R_TRIG_1(CLK := hmi_Manual_cal); // R_TRIG
Corrected_count := _w1;
Zero_count := _w2;
Zero_depth_count := Roll_over_count / 2;
IF _w3 THEN (* Corrected_count + Roll_over_count; result not used *) END_IF
IF Corrected_count > (Roll_over_count - Zero_depth_count) THEN (* Corrected_count - Roll_over_count; result not used *) END_IF
R_TRIG_0(CLK := Manual_cal); // R_TRIG
IF R_TRIG_0.Q OR R_TRIG_1.Q THEN _w2 := Count; END_IF
_w1 := Count - Zero_count;
_w3 := Corrected_count < (-Zero_depth_count);
END_METHOD

METHOD M_Depth_history
VAR_INPUT
END_VAR
VAR_INST // added by the converter: edge detectors and wires of the graphical bodies
    _w1, _w2, _w6, _w7 : REAL;
    _w3, _w4 : ANY;
    _w5, _w8 : BOOL;
END_VAR
IF New_depth THEN _w1 := Raw_depth; END_IF
Scan_count := _w2;
IF Late_depth THEN _w3 := 1; END_IF
IF New_depth THEN _w4 := ROL(Depth_history, 1); END_IF
Late_depth := _w5;
_w6 := Raw_depth;
Scan_count := _w7;
New_depth := _w8;
Raw_depth_prev := _w3;
IF NOT New_depth THEN _w2 := Raw_depth + Raw_depth_prev; END_IF
IF New_depth THEN _w7 := 0; END_IF
Depth_history[0] := _w1;
_w5 := Scan_count = Scans_per_update;
_w8 := Raw_depth <> Raw_depth_prev;
Raw_depth_prev := _w6;
Depth_history := _w4;
END_METHOD

METHOD M_Direction
VAR_INPUT
END_VAR
VAR_INST // added by the converter: edge detectors and wires of the graphical bodies
    _w1, _w2, _w3 : REAL;
    _w4, _w5, _w6, _w7, _w9 : BOOL;
    _w8, _w10 : ANY;
END_VAR
Max_pos_reached := _w1;
Max_pos_reached := _w2;
_w3 := Max_pos_reached + Direction_hysteresis;
_w4 := Raw_depth > Max_pos_reached;
IF Going_up AND _w5 THEN _w1 := Raw_depth; END_IF
_w5 := Raw_depth < Max_pos_reached;
_w7 := Going_up AND _w6;
_w6 := Raw_depth > _w3;
IF NOT Going_up AND _w4 THEN _w2 := Raw_depth; END_IF
SR_0(SET1 := _w8, RESET := _w7); // SR
_w8 := NOT Going_up AND _w9;
_w9 := Raw_depth < _w10;
Going_up := SR_0.Q1;
_w10 := Max_pos_reached - Direction_hysteresis;
END_METHOD

METHOD M_Encoder_cal
VAR_INPUT
END_VAR
VAR_INST // added by the converter: edge detectors and wires of the graphical bodies
    _w1, _w3, _w6 : REAL;
    _w2, _w9, _w10, _w11 : ANY;
    _w4, _w5, _w7, _w8 : BOOL;
END_VAR
_w1 := Cal_switch_depth + Cal_window_down;
Offset := _w3;
_w5 := _w4 AND Calibrate AND NOT Rope_capping_mode;
Open_below := Raw_depth > _w2 AND NOT Calibrate AND NOT Rope_capping_mode;
F_TRIG_0(CLK := Calibrate); // F_TRIG
IF F_TRIG_0.Q THEN _w6 := Raw_depth; END_IF
Closed_above := _w5;
Captured_depth := _w6;
_w8 := Captured_depth >= Cal_switch_depth - Cal_window_up AND F_TRIG_0.Q AND _w7 AND NOT Disallow_multiple_cal;
_w7 := Captured_depth <= _w1;
IF _w8 THEN _w3 := _w9; END_IF
_w9 := Cal_switch_depth - Captured_depth;
_w2 := Cal_switch_depth + Cal_window_down;
RS_0(SET := F_TRIG_0.Q, RESET1 := _w10); // RS
_w10 := Raw_depth > _w1;
_w4 := Raw_depth < _w11;
_w11 := Cal_switch_depth - Cal_window_up;
Disallow_multiple_cal := RS_0.Q1;
END_METHOD

METHOD M_Encoder_depth
VAR_INPUT
END_VAR
VAR_INST // added by the converter: edge detectors and wires of the graphical bodies
    _w1, _w2, _w4 : BOOL;
    _w3, _w6, _w7 : REAL;
    _w5 : ANY;
END_VAR
_w2 := ((-Offset) > Cal_window_up OR _w1) + NOT Rope_capping_mode;
_w3 := Raw_depth + Offset;
_w4 := Raw_depth > Max_depth;
Raw_depth := _w6;
Raw_depth := _w5 + NOT Rope_capping_mode;
Encoder_mm := _w7;
_w6 := Encoder_mm + Manual_cal_depth;
_w1 := Offset > Cal_window_down;
_w5 := Min_depth > Raw_depth OR _w4;
Offset_out_of_range := _w2;
Raw_depth := LIMIT(Min_depth, Raw_depth, Max_depth);
_w7 := Corrected_count * mm_per_count;
Calibrated_depth := _w3;
END_METHOD

METHOD M_HMI_command
VAR_INPUT
END_VAR
FB_WORD_TO_BIT_V0_0(Word_in := hmi_Data.Status); // FB_WORD_TO_BIT_V0
hmi_Manual_cal := FB_WORD_TO_BIT_V0_0.bit0;
END_METHOD

METHOD M_HMI_data
VAR_INPUT
END_VAR
VAR_INST // added by the converter: edge detectors and wires of the graphical bodies
    _w1, _w2 : REAL;
    _w3 : ANY;
END_VAR
hmi_data.Status := FB_BIT_TO_WORD_V0_0.Word_out;
_w1 := Count;
_w2 := Raw_depth;
FB_BIT_TO_WORD_V0_0(bit1 := Going_up, bit2 := Movement_detect, bit3 := Calibrate); // FB_BIT_TO_WORD_V0
hmi_data.Calibrated_depth := _w3;
hmi_data.Status := _w1;
hmi_data.Compensated_depth := Compensated_depth;
hmi_data.Raw_depth := _w2;
_w3 := Calibrated_depth;
hmi_data.Raw_count := Raw_count;
hmi_data.Speed := Speed;
END_METHOD

METHOD M_Layering_compensation
VAR_INPUT
END_VAR
VAR_INST // added by the converter: edge detectors and wires of the graphical bodies
    _w1 : REAL;
    _w2 : ANY;
END_VAR
Compensation := _w1;
_w1 := _w2 * Mid_wind_error;
// Add the compensation to the calibrated depth.
Compensated_depth := Calibrated_depth + Compensation;
// Calculate approximate error caused by rope layering. The error should be calibrated to zero at Wind_top_depth and Wind_bottom depth.
// The maximum error should occur roughly at mid-wind (Mid_wind_error). The error is approximated using a sine function.
_w2 := SIN(((Calibrated_depth - Wind_top_depth) / (Wind_bottom_depth - Wind_top_depth)) * 3.14159265);
END_METHOD

METHOD M_Movement_detect
VAR_INPUT
END_VAR
VAR_INST // added by the converter: edge detectors and wires of the graphical bodies
    _w1 : ANY;
    _w2 : REAL;
END_VAR
Movement_detect := RS_1.Q1;
TON_0(IN := Brakes_proved_on, PT := t#500ms); // TON
Brakes_proved_on_500ms := TON_0.Q;
RS_1(SET := ABS(Raw_depth - Brakes_on_depth) > Movement_detect_dist, RESET1 := _w1); // RS
R_TRIG_2(CLK := Brakes_proved_on_500ms); // R_TRIG
_w1 := R_TRIG_2.Q OR Winder_reset;
IF _w1 THEN _w2 := Raw_depth; END_IF
Brakes_on_depth := _w2;
END_METHOD

METHOD M_Speed
VAR_INPUT
END_VAR
VAR
	fbGetCurTaskIdx  : GETCURTASKINDEX;
END_VAR
{warning 'TODO: Task info cycle time is being converted from UDINT to REAL with possible data loss.'}
Speed := (Depth_history[0] - Depth_history[Speed_ave_intervals]) * 1000 
	/ (_TaskInfo[fbGetCurTaskIdx.index].CycleTime * Scans_per_update * Speed_ave_intervals);
END_METHOD

END_FUNCTION_BLOCK

// ---- POUs/FBs/FB_Fast_brake.TcPOU
FUNCTION_BLOCK FB_Fast_brake
VAR_INPUT
	Lh_depth:REAL;
	Rh_depth:REAL;
	Speed:REAL;
	Fast_brake_top_depth:REAL;
	Fast_brake_bottom_depth:REAL;
	Fast_brake_speed:REAL;
	Speed_hysteresis:REAL;
	Off_delay_after_brakes_on:TIME;
	Check_speed:REAL;
END_VAR
VAR_OUTPUT
	Valve:BOOL;
	Active_above_check_speed:BOOL;
END_VAR
VAR
	FB_CTRL_HYSTERESIS_0: FB_CTRL_HYSTERESIS;
	TON_0: TON;
END_VAR

M_Fast_brake();

METHOD M_Fast_brake
VAR_INPUT
END_VAR
{warning 'TODO: HYSTERESIS block needs to be figured out and made to work correctly.'}
VAR_INST // added by the converter: edge detectors and wires of the graphical bodies
    _w1, _w2, _w3, _w4, _w5, _w7 : BOOL;
    _w6 : ANY;
END_VAR
_w1 := Rh_depth <= Fast_brake_top_depth;
_w2 := Lh_depth >= Fast_brake_bottom_depth;
// Lockout if fast brake valve is enabled above check speed
_w3 := Rh_depth >= Fast_brake_bottom_depth;
Active_above_check_speed := (ABS(Speed)) >= Check_speed AND Valve;
_w6 := _w4 AND NOT TON_0.Q AND NOT _w5;
_w5 := (ABS(Speed)) >= 300;
TON_0(IN := Brakes.Proved_on, PT := Off_delay_after_brakes_on); // TON
// Fast braking
FB_CTRL_HYSTERESIS_0(); // FB_CTRL_HYSTERESIS
_w4 := NOT FB_CTRL_HYSTERESIS_0.bOut AND Safety.Sc1 AND Safety.Sc2 OR NOT Clutch.Lh_in OR NOT Clutch.Rh_in OR _w7 OR _w1 OR _w2 OR _w3;
Valve := _w6;
_w7 := Lh_depth <= Fast_brake_top_depth;
END_METHOD

END_FUNCTION_BLOCK

// ---- POUs/FBs/FB_Least_gate_element.TcPOU
FUNCTION_BLOCK FB_Least_gate_element
VAR_INPUT
	Enforce:BOOL;
	Enforce_in_rope_cap:BOOL;
	Allowed_speed:REAL;
	Description:STRING[32];
END_VAR
VAR_OUTPUT
END_VAR
VAR_IN_OUT
	Least_gate_data:dut_Least_gate;
END_VAR
VAR
END_VAR

M_Least_gate_element();

METHOD M_Least_gate_element
VAR_INPUT
END_VAR
VAR_INST // added by the converter: edge detectors and wires of the graphical bodies
    _w1, _w4, _w5 : BOOL;
    _w2, _w3 : ANY;
    _w6 : REAL;
END_VAR
IF _w1 THEN _w2 := Description; END_IF
_w4 := Allowed_speed < _w3;
_w3 := BOOL_TO_REAL(Least_gate_data.Rope_cap_mode);
_w1 := _w4 AND Enforce AND NOT _w5;
IF _w1 THEN _w6 := Allowed_speed; END_IF
Least_gate_data.Min_allowed_speed := _w6;
_w5 := Least_gate_data.Rope_cap_mode AND NOT Enforce_in_rope_cap;
Least_gate_data.Description := _w2;
END_METHOD

END_FUNCTION_BLOCK

// ---- POUs/FBs/FB_Least_gate_result.TcPOU
FUNCTION_BLOCK FB_Least_gate_result
VAR_INPUT
	Rope_cap_mode:BOOL;
END_VAR
VAR_OUTPUT
	Allowed_speed:REAL;
	Description:STRING[32];
END_VAR
VAR_IN_OUT
	Least_gate_data:dut_Least_gate;
END_VAR
VAR
END_VAR

M_Least_gate_result();

METHOD M_Least_gate_result
VAR_INPUT
END_VAR
VAR_INST // added by the converter: edge detectors and wires of the graphical bodies
    _w1, _w2 : ANY;
END_VAR
Least_gate_data.Min_allowed_speed := _w1;
Description := _w2;
_w2 := Least_gate_data.Description;
_w1 := 32000;
Allowed_speed := Least_gate_data.Min_allowed_speed;
Least_gate_data.Description := '';
Least_gate_data.Rope_cap_mode := Rope_cap_mode;
END_METHOD

END_FUNCTION_BLOCK

// ---- POUs/FBs/FB_Mode.TcPOU
FUNCTION_BLOCK FB_Mode
VAR_INPUT
	Men:BOOL;
	Material:BOOL;
	Rock:BOOL;
	Manual_switch:BOOL;
	Auto_switch:BOOL;
	Rope_capping_switch:BOOL;
	Brake_maint_switch:BOOL;
	Single_lever_control:BOOL;
END_VAR
VAR_OUTPUT
	cs_Mode_change:BOOL;
	cs_Men_rock_sw_fault:BOOL;
	cs_Auto_manual_sw_fault:BOOL;
	cs_Men_to_rock:BOOL;
	cs_Rock_to_men:BOOL;
	cs_Auto_to_manual:BOOL;
	cs_Manual_to_auto:BOOL;
	cs_Rope_capping_on:BOOL;
	cs_Rope_capping_off:BOOL;
	cs_Brake_maint_on:BOOL;
	cs_Brake_maint_off:BOOL;
	hmi_Status:WORD;
END_VAR
VAR
	F_TRIG_0: F_TRIG;
	R_TRIG_0: R_TRIG;
	R_TRIG_1: R_TRIG;
	F_TRIG_1: F_TRIG;
	R_TRIG_2: R_TRIG;
	F_TRIG_2: F_TRIG;
	R_TRIG_3: R_TRIG;
	F_TRIG_3: F_TRIG;
	R_TRIG_4: R_TRIG;
	F_TRIG_4: F_TRIG;
	R_TRIG_5: R_TRIG;
	F_TRIG_5: F_TRIG;
	TON_0: TON;
	BIT_TO_WORD_V0_0: FB_BIT_TO_WORD_V0;
END_VAR

M_Mode();
M_Mode_faults();

METHOD M_Mode
VAR_INPUT
END_VAR

VAR
END_VAR
// Mode section
Mode.Men := Men AND NOT Material AND NOT Rock;
Mode.Rope_capping := Rope_capping_switch;
BIT_TO_WORD_V0_0(
    bit0 := Mode.Manual,
    bit1 := Mode.Auto,
    bit2 := Mode.Auto_go,
    bit3 := Mode.Men,
    bit4 := Mode.Material,
    bit5 := Mode.Rock,
    bit6 := Mode.Rope_capping,
    bit7 := Mode.Brake_maintenance,
    bit8 := Mode.Auto_switch,
    bit9 := Mode.Single_lever_control); // FB_BIT_TO_WORD_V0
Mode.Brake_maintenance := Brake_maint_switch;
Mode.Material := NOT Men AND Material AND NOT Rock;
Mode.Auto_switch := Auto_switch;
Mode.Rock := NOT Men AND NOT Material AND Rock;
hmi_Status := BIT_TO_WORD_V0_0.Word_out;
Mode.Single_lever_control := Single_lever_control;
Mode.Manual := Manual_switch AND NOT Auto_switch;
END_METHOD

METHOD M_Mode_faults
VAR_INPUT
END_VAR
VAR_INST // added by the converter: edge detectors and wires of the graphical bodies
    _w1, _w2, _w3 : BOOL;
END_VAR
// Mode faults section
// Fault to trip winder on any state of change on switches
// The TRIGGER FB does not exist in Codesys so I am using a rising and falling trigger for each function.
R_TRIG_0(CLK := Men); // R_TRIG
(* R_TRIG_0.Q OR F_TRIG_0.Q OR R_TRIG_1.Q OR F_TRIG_1.Q OR R_TRIG_1.Q OR F_TRIG_1.Q OR R_TRIG_2.Q OR F_TRIG_2.Q OR R_TRIG_3.Q OR F_TRIG_3.Q OR R_TRIG_4.Q OR F_TRIG_4.Q OR R_TRIG_5.Q OR F_TRIG_5.Q; result not used *)
F_TRIG_0(CLK := Men); // F_TRIG
cs_Rock_to_men := R_TRIG_0.Q OR F_TRIG_1.Q;
R_TRIG_1(CLK := Material); // R_TRIG
F_TRIG_1(CLK := Material); // F_TRIG
cs_Men_to_rock := F_TRIG_0.Q OR R_TRIG_1.Q;
R_TRIG_1(CLK := Rock); // R_TRIG
F_TRIG_1(CLK := Rock); // F_TRIG
R_TRIG_2(CLK := Manual_switch); // R_TRIG
cs_Auto_to_manual := R_TRIG_2.Q;
F_TRIG_2(CLK := Manual_switch); // F_TRIG
R_TRIG_3(CLK := Auto_switch); // R_TRIG
cs_Manual_to_auto := R_TRIG_3.Q;
F_TRIG_3(CLK := Auto_switch); // F_TRIG
R_TRIG_4(CLK := Rope_capping_switch); // R_TRIG
cs_Rope_capping_on := R_TRIG_4.Q;
F_TRIG_4(CLK := Rope_capping_switch); // F_TRIG
cs_Rope_capping_off := F_TRIG_4.Q;
R_TRIG_5(CLK := Brake_maint_switch); // R_TRIG
cs_Brake_maint_on := R_TRIG_5.Q;
F_TRIG_5(CLK := Brake_maint_switch); // F_TRIG
cs_Brake_maint_off := F_TRIG_5.Q;
// Men Material Rock switch fault
TON_0(IN := NOT (Men AND NOT Material AND NOT Rock) AND NOT _w1 AND NOT _w2, PT := t#200ms); // TON
cs_Men_rock_sw_fault := TON_0.Q;
_w1 := NOT Men AND Material AND NOT Rock;
_w2 := NOT Men AND NOT Material AND Rock;
// Auto Manual switch fault
cs_Auto_manual_sw_fault := NOT (Auto_switch AND NOT Manual_switch) AND NOT _w3;
_w3 := NOT Auto_switch AND Manual_switch;
END_METHOD

END_FUNCTION_BLOCK

// ---- POUs/FBs/FB_Moving_average.TcPOU
FUNCTION_BLOCK FB_Moving_average
VAR_INPUT
	New_sample: REAL;
	Num_samples: INT;
END_VAR
VAR_OUTPUT
	Out: REAL;
END_VAR
VAR CONSTANT
	Array_size: INT := 300;	
END_VAR
VAR
	Samples: ARRAY[0..(Array_size - 1)] OF REAL;
	i: INT;
	Sum: REAL;
END_VAR

Sum:= 0;
FOR i :=

END_FUNCTION_BLOCK

// ---- POUs/FBs/FB_Power_lever.TcPOU
FUNCTION_BLOCK FB_Power_lever
VAR_INPUT
	Forward:BOOL; (*Lever notch 1 forward*)
	Reverse:BOOL; (*Lever notch 1 reverse*)
	Pot:INT; (*Analogue value from lever potentiometer*)
	Button:BOOL;
	Neutral:BOOL; 
	Use_neutral:BOOL;
	Fully_fwd_val:INT; (*Value of analogue input when lever is fully forward*)
	Neutral_val:INT; (*Value of analogue input when lever is in neutral*)
	Fully_rev_val:INT; (*Value of analogue input when lever is fully reverse*)
	Zero_deadband:REAL; (*Lever zero position deadband on a scale of 0 to 100.0 i.e. a value of 1 gives a 1% deadband in each direction*)
	Full_lever_deadband:REAL; (*Lever fully forward or reverse deadband on a scale of 0 to 100.0 i.e. a value of 100 gives a 1% deadband*)
	Notch_position:REAL; (*Lever value (-100.0 to 100.0, no deadbands) at which forward and reverse notches change state*)
	Allowed_notch_variation:REAL; (*Allowed variation in notch position*)
	Pos_out_of_range_val:INT; (*If the analogue Pot value exceeds this threshold, a fault will be generated.*)
	Neg_out_of_range_val:INT; (*If the analogue Pot value is less than this threshold, a fault will be generated.*)
END_VAR
VAR_OUTPUT
	Raw:REAL; (*Linear scaled lever value with no deadbands applied. -10 000 = fully reverse. +10 000 = fully forward.*)
	Linear:REAL; (*Linear scaled lever value with deadbands applied. -10 000 = fully reverse. +10 000 = fully forward.*)
	Cubic:REAL; (*Cubic scaling applied to lever value with deadbands applied. -10 000 = fully reverse. +10 000 = fully forward.*)
	cs_Forward_and_reverse:BOOL; (*Forward and reverse inputs both energised.*)
	cs_Pot_fwd_no_notch:BOOL; (*Pot shows that lever is forward but the forward notch is not activated*)
	cs_Pot_rev_no_notch:BOOL; (*Pot shows that lever is reverse but the reverse notch is not activated*)
	cs_Fwd_notch_not_pot:BOOL; (*Reverse notch is activated but the pot does not show that the lever is past the reverse notch*)
	cs_Rev_notch_not_pot:BOOL; (*Forward notch is activated but the pot does not show that the lever is past the forward notch*)
	cs_Out_of_range_pos:BOOL; (*The Pot value is out of range in the positive direction*)
	cs_Out_of_range_neg:BOOL; (*The Pot value is out of range in the negative direction*)
	hmi_data:dut_hmi_Power_lever; (*HMI status bits as well as Raw, Linear and Cubic values*)
END_VAR
VAR
	Linear_abs: INT;
	hmi_Word:WORD;
	TON_0: TON;
	TON_2: TON;
	TON_1: TON;
	TON_3: TON;
	BIT_TO_WORD_V0_0: FB_BIT_TO_WORD_V0;
END_VAR

M_Lever_scaling();
M_Power_lever_data();
M_Power_lever_faults();

METHOD M_Lever_scaling
VAR_INPUT
END_VAR
VAR_INST // added by the converter: edge detectors and wires of the graphical bodies
    _w1, _w2, _w3, _w4, _w5, _w6 : ANY;
END_VAR
// Lever scaling section
// Scale Drivers Lever reference to compensate for Voltage input that is not exactly +/-10V.
Raw := ((INT_TO_REAL(Pot) - _w1) * 200.0) / _w2;
_w1 := (_w4 + _w5) / 2.0;
_w4 := INT_TO_REAL(Fully_fwd_val);
_w2 := _w4 - _w5;
_w5 := INT_TO_REAL(Fully_rev_val);
// Apply deadbands to absolute value.
Linear_abs := _w3 / (100.0 - Zero_deadband - Full_lever_deadband);
_w3 := (ABS(Raw) - Zero_deadband) * 100.0;
// Limit ouput to max of 10000
Linear_abs := LIMIT(0.0, Linear_abs, 100.0);
// Add sign back to the absolute value.
Linear := SEL(Raw >= 0, -Linear_abs, Linear_abs);
// Apply cubic function
Cubic := (Linear * Linear * Linear) / _w6;
_w6 := 100.0 * 100.0;
END_METHOD

METHOD M_Power_lever_data
VAR_INPUT
END_VAR

VAR
END_VAR
// Power lever data section
// Pack data in Power_lever_data stucture.
Power_lever.Forward := SEL(Use_neutral, Forward, Linear > 0 AND NOT Neutral);
Power_lever.Reverse := SEL(Use_neutral, Reverse, Linear < 0 AND NOT Neutral);
// Pack data for HMI
BIT_TO_WORD_V0_0(
    bit0 := Power_lever.Forward,
    bit1 := Power_lever.Reverse,
    bit2 := Power_lever.Neutral,
    bit3 := Button); // FB_BIT_TO_WORD_V0
hmi_Data.Status := BIT_TO_WORD_V0_0.Word_out;
Power_lever.Button := Button;
Power_lever.Raw := Raw;
Power_lever.Linear := Linear;
Power_lever.Cubic := Cubic;
hmi_data.Raw := Raw;
Power_lever.Neutral := Neutral AND Use_neutral OR Forward AND Reverse AND NOT Use_neutral;
hmi_data.Linear := Linear;
hmi_data.Cubic := Cubic;
END_METHOD

METHOD M_Power_lever_faults
VAR_INPUT
END_VAR
VAR_INST // added by the converter: edge detectors and wires of the graphical bodies
    _w1, _w2, _w3, _w4 : ANY;
END_VAR
// Power lever faults section
// Forward and reverse notches simulateously active
cs_Forward_and_reverse := Forward AND Reverse;
TON_0(IN := Raw > _w1 AND NOT Forward, PT := t#500ms); // TON
// Pot shows that lever is forward but the forward notch is not activated
_w1 := Notch_position + Allowed_notch_variation;
cs_Pot_fwd_no_notch := TON_0.Q;
TON_1(IN := (-Raw) > _w2 AND NOT Reverse, PT := t#500ms); // TON
// Pot shows that lever is reverse but the reverse notch is not activated
_w2 := Notch_position + Allowed_notch_variation;
cs_Pot_rev_no_notch := TON_1.Q;
TON_2(IN := Raw < _w3 AND Forward, PT := t#500ms); // TON
// Forward notch is activated but the pot does not show that the lever is past the forward notch
_w3 := Notch_position - Allowed_notch_variation;
cs_Fwd_notch_not_pot := TON_2.Q;
TON_3(IN := (-Raw) < _w4 AND Reverse, PT := t#500ms); // TON
// Reverse notch is activated but the pot does not show that the lever is past the reverse notch
_w4 := Notch_position - Allowed_notch_variation;
cs_Rev_notch_not_pot := TON_3.Q;
// Pot is out of range positive
cs_Out_of_range_pos := Pot > Pos_out_of_range_val;
// Pot is out of range negative
cs_Out_of_range_neg := Pot < Neg_out_of_range_val;
END_METHOD

END_FUNCTION_BLOCK

// ---- POUs/FBs/FB_Standard_stuff.TcPOU
FUNCTION_BLOCK FB_Standard_stuff
VAR_INPUT
	Bits_from_hmi:ARRAY[0..1] OF WORD;
	Creep_switch:BOOL;
	Slow_switch:BOOL;
	Normal_switch:BOOL;
	Watchdog_heartbeat:BOOL;
	System_start:BOOL;
	System_stop:BOOL;
	System_started:BOOL;
END_VAR
VAR_OUTPUT
	Bits_to_hmi:ARRAY[0..1] OF WORD;
	Hmi_test_trip:BOOL;
	Watchdog_test_0:BOOL;
	Watchdog_test_1:BOOL;
	Activity:BOOL;
END_VAR

// Standard Stuff section
// Word to Bit and Bit to Word don't exist in the form we need them so I pack this manually using address references.
Hmi_test_trip := Bits_from_hmi[0].0;
Bits_to_hmi[0].0 := Creep_switch;
Watchdog_test_0 := Bits_from_hmi[0].1;
Bits_to_hmi[0].1 := Slow_switch;
Watchdog_test_1 := Bits_from_hmi[0].2;
Bits_to_hmi[0].2 := Normal_switch;
Activity := Bits_from_hmi[0].3;
Bits_to_hmi[0].3 := Watchdog_heartbeat;
Bits_to_hmi[0].4 := System_start;
Bits_to_hmi[0].5 := System_stop;
Bits_to_hmi[0].6 := System_started;

END_FUNCTION_BLOCK

// ---- POUs/FBs/FB_Torque_prediction.TcPOU
FUNCTION_BLOCK FB_Torque_prediction
VAR_INPUT
	Lh_depth:REAL;
	Rh_depth:REAL;
	Levels:ARRAY[0..31]OF REAL;
	Bottom_level:REAL;
	Enable:BOOL;
	Lh_full_load:BOOL;
	Lh_half_load:BOOL;
	Rh_full_load:BOOL;
	Rh_half_load:BOOL;
	Speed_ref:REAL;
	Speed:REAL;
	Speed_control:BOOL;
END_VAR
VAR_OUTPUT
	Predicted_current:REAL;
END_VAR
VAR
	Speed_ref_prev:REAL;
	Speed_ramp_rate:REAL;
	Moving_fwd:BOOL;
	Moving_rev:BOOL;
	Rev_pulse:BOOL;
	Fwd_pulse:BOOL;
	FB_LAG_FILTER_0: FB_Lag_filter;
	RS_0: RS;
	RS_1: RS;
	FB_TP_with_stop_0: FB_TP_with_stop;
	FB_TP_with_stop_1: FB_TP_with_stop;
END_VAR

M_Torque_prediction();

END_FUNCTION_BLOCK

// ---- POUs/FBs/FB_TP_with_stop.TcPOU
FUNCTION_BLOCK FB_TP_with_stop
VAR_INPUT
	Start:BOOL;
	Stop:BOOL;
	PT:TIME;
END_VAR
VAR_OUTPUT
	Q:BOOL;
	ET:TIME;
END_VAR
VAR
	R_TRIG_0: R_TRIG;
	TON_0: TON;
	RS_0: RS;
END_VAR

M_TP_with_stop();

METHOD M_TP_with_stop
VAR_INPUT
END_VAR
VAR_INST // added by the converter: edge detectors and wires of the graphical bodies
    _w1 : BOOL;
END_VAR
Q := RS_0.Q1;
_w1 := TON_0.Q OR Stop;
R_TRIG_0(CLK := Start); // R_TRIG
RS_0(SET := R_TRIG_0.Q, RESET1 := _w1); // RS
TON_0(IN := Start, PT := PT); // TON
END_METHOD

END_FUNCTION_BLOCK

// ---- POUs/FBs/FB_Torque_prediction_ST.TcPOU
FUNCTION_BLOCK FB_Torque_prediction_ST
VAR_INPUT
END_VAR
VAR_OUTPUT
END_VAR
VAR
	Lh_full: BOOL;
	Lh_half: BOOL;
	Equal: BOOL;
	Rh_half: BOOL;
	Rh_full: BOOL;
	
	Lh_full_selected: BOOL;
	Lh_half_selected: BOOL;
	Equal_selected: BOOL;
	Rh_half_selected: BOOL;
	Rh_full_selected: BOOL;
	
	R_TRIG0: R_TRIG;
	R_TRIG1: R_TRIG;
	R_TRIG2: R_TRIG;
	R_TRIG3: R_TRIG;
	R_TRIG4: R_TRIG;
END_VAR

R_TRIG0(CLK:= Torque_prediction.Lh_full_request, Q=> Lh_full_selected);
R_TRIG1(CLK:= Torque_prediction.Lh_half_request, Q=> Lh_half_selected);
R_TRIG2(CLK:= Torque_prediction.Equal_request, Q=> Equal_selected);
R_TRIG3(CLK:= Torque_prediction.Rh_half_request, Q=> Rh_half_selected);
R_TRIG4(CLK:= Torque_prediction.Rh_full_request, Q=> Rh_full_selected);

IF Lh_full_selected THEN
	Torque_prediction.Lh_full := 1;
	Torque_prediction.Lh_half := 0;
	Torque_prediction.Equal := 0;
	Torque_prediction.Rh_half := 0;
	Torque_prediction.Rh_full := 0;
ELSIF Lh_half_selected THEN
	Torque_prediction.Lh_full := 0;
	Torque_prediction.Lh_half := 1;
	Torque_prediction.Equal := 0;
	Torque_prediction.Rh_half := 0;
	Torque_prediction.Rh_full := 0;
ELSIF Equal_selected THEN
	Torque_prediction.Lh_full := 0;
	Torque_prediction.Lh_half := 0;
	Torque_prediction.Equal := 1;
	Torque_prediction.Rh_half := 0;
	Torque_prediction.Rh_full := 0;
ELSIF Rh_half_selected THEN
	Torque_prediction.Lh_full := 0;
	Torque_prediction.Lh_half := 0;
	Torque_prediction.Equal := 0;
	Torque_prediction.Rh_half := 1;
	Torque_prediction.Rh_full := 0;
ELSIF Rh_full_selected THEN
	Torque_prediction.Lh_full := 0;
	Torque_prediction.Lh_half := 0;
	Torque_prediction.Equal := 0;
	Torque_prediction.Rh_half := 0;
	Torque_prediction.Rh_full := 1;
END_IF

Torque_prediction.Lh_full_request := 0;
Torque_prediction.Lh_half_request := 0;
Torque_prediction.Equal_request := 0;
Torque_prediction.Rh_half_request := 0;
Torque_prediction.Rh_full_request := 0;

END_FUNCTION_BLOCK

// ---- POUs/FBs/FB_TPD_CANopen.TcPOU
FUNCTION_BLOCK FB_TPD_CANopen
VAR_INPUT
	Node_address:STRING; (*CANopen node address of DCV*)
	Enable:BOOL;
	Start:BOOL;
	Reset:BOOL;
	Torque_control:BOOL;
	Speed_ref:REAL; (*Speed ref in m/s (with drive ramp)*)
	Torque_ref:REAL; (*Torque ref  in Amps for DC or as a percent of full load current for AC*)
	Nominal_speed:REAL; (*Speed in m/s at rated motor rpm*)
	Current_limit_P:REAL;
	Current_limit_N:REAL;
	Speed_P:REAL;
	Speed_I:REAL;
	Write_config:BOOL;
	Check_config:BOOL;
	Base_settings:dut_TPD32_base_settings;
	Status_word:REAL; (*DCV status word - adheres to DRIVECOM standard - same as ATV71*)
	PDO_TX1:REAL; (*DCV transmit PDO 1*)
	PDO_TX2:REAL; (*DCV transmit PDO 2*)
	PDO_TX3:REAL; (*DCV transmit PDO 3*)
END_VAR
VAR_OUTPUT
	Running:BOOL; (*Drive enabled and operational - from Control Word*)
	Fault:BOOL; (*Drive is reporting a malfunction*)
	hmi_Motor_speed:dut_hmi_Analogue; (*Motor speed in rpm*)
	hmi_Amature_current:dut_hmi_Analogue; (*Armature current as % of full load current*)
	hmi_Field_current:dut_hmi_Analogue; (*Field current as % of nominal field current*)
	hmi_Amature_voltage:dut_hmi_Analogue; (*Armature voltage in volts*)
	Mains_failure:BOOL;
	Field_failure:BOOL;
	Configuring:BOOL;
	Config_mismatch:BOOL;
	Virt_dig_in:REAL; (*DCV virtual digital inputs*)
	PDO_RX1:REAL; (*DCV receive PDO 1*)
	PDO_RX2:REAL; (*DCV receive PDO 2*)
	PDO_RX3:REAL; (*DCV receive PDO 3*)
END_VAR
VAR
	GEST1:ARRAY[1..4]OF REAL;
	Node_addm:ARRAY[0..8]OF REAL;
	Topo_address:STRING;
	Flux_current_array:ARRAY[1..2]OF REAL;
	i:REAL;
	Motor_speed:REAL;
	Amature_current:REAL;
	Amature_voltage:REAL;
	Field_current:REAL;
END_VAR
{warning 'TODO: Var Status_word was set as an INT in the original program. I have set it as a REAL as per our current structure, but should this not be a word?'}
{warning 'TODO: This function block needs to be reworked to work on our new comms'}

M_DCV_PDO();
M_DCV_config();
M_Settings();
M_DCV_analogues();

METHOD M_DCV_PDO
VAR_INPUT
END_VAR
{warning 'TODO: these comms need to be recreated as EtherCat comms I assume? The ADDM FB doesn't exist here.'}
VAR_INST // added by the converter: edge detectors and wires of the graphical bodies
    _w1 : STRING;
END_VAR
Topo_address := _w1;
// Convert Node address to topological address for SDO reads/writes
_w1 := CONCAT(STR1 := '0.0.2', STR2 := Node_address);
END_METHOD

END_FUNCTION_BLOCK

// ---- POUs/FBs/FB_Trip_control.TcPOU
FUNCTION_BLOCK FB_Trip_control
VAR_INPUT
	Category:REAL;
	First_up:BOOL;
	Fault0:BOOL;
	Fault1:BOOL;
	Fault2:BOOL;
	Fault3:BOOL;
	Fault4:BOOL;
	Fault5:BOOL;
	Fault6:BOOL;
	Fault7:BOOL;
	Fault8:BOOL;
	Fault9:BOOL;
	Fault10:BOOL;
	Fault11:BOOL;
	Fault12:BOOL;
	Fault13:BOOL;
	Fault14:BOOL;
	Fault15:BOOL;
	Reset:BOOL;
	Inhibit:BOOL;
	Block_ID:REAL;
END_VAR
VAR_OUTPUT
	Trip_present:BOOL;
	Trip0:BOOL;
	Trip1:BOOL;
	Trip2:BOOL;
	Trip3:BOOL;
	Trip4:BOOL;
	Trip5:BOOL;
	Trip6:BOOL;
	Trip7:BOOL;
	Trip8:BOOL;
	Trip9:BOOL;
	Trip10:BOOL;
	Trip11:BOOL;
	Trip12:BOOL;
	Trip13:BOOL;
	Trip14:BOOL;
	Trip15:BOOL;
END_VAR
VAR_IN_OUT
END_VAR
VAR
END_VAR
{warning 'TODO: Trip_control has not been done and needs to be gone over with Bret.'}

END_FUNCTION_BLOCK

// ---- POUs/Sections/Winder_data.TcPOU
PROGRAM Winder_data
VAR
	TP_0: TP;
	TP_1: TP;
	TP_2: TP;
	Power_lever_0: FB_Power_lever;
	Clutch_0: FB_Clutch;
	Mode_0: FB_Mode;
	Brake_0: FB_Brake;
	Standard_stuff_0: FB_Standard_stuff;
END_VAR

// Safety data
// Power lever
Power_lever_0(); // FB_Power_lever
// Clutch data
Clutch_0(); // FB_Clutch
// Brake data
Brake_0(); // Brake
// Mode data
Mode_0(); // FB_Mode
// Standard bits
Standard_stuff_0(); // FB_Standard_stuff

END_PROGRAM
